DATA_BLOCK "HmiDb"
{ S7_Optimized_Access := 'TRUE' }
AUTHOR : Searinox
VERSION : 0.1
NON_RETAIN
"Hmi"

BEGIN

END_DATA_BLOCK

